Staubli VAL3: startingSockets.pgx

program startingSockets()
begin
  clearBuffer(sSocket)
  //clearBuffer(sPlc)
  wait(sioSet(sSocket, 73)==1)
  //wait(sioGet(sPlc, nRecvPLC)==1)

end
